INTERFACE I_StateMachine EXTENDS I_Debug

METHOD Change : Result
VAR_INPUT
	iNewState	: I_StateInternal;
END_VAR
VAR_OUTPUT
	iOldState	: I_StateInternal;
END_VAR
END_METHOD

END_INTERFACE

(* stored: Version 1.1.0.1
   Itf I_StateMachine: Id {9c44ba60-8196-4755-9ee3-5f232b421b4a}
   Method Change: Id {37759f66-045e-4326-b96d-cd069d93483c} *)
